FUNCTION FC_Concat4 : STRING
VAR_INPUT
    STR1: STRING(255);
    STR2: STRING(255);
    STR3: STRING(255):= '';
    STR4: STRING(255):= '';
    // etc up to a large number
END_VAR
VAR
	
END_VAR



FC_Concat4 := CONCAT(STR1 := FC_Concat4, STR2 := STR1);
FC_Concat4 := CONCAT(STR1 := FC_Concat4, STR2 := STR2);
FC_Concat4 := CONCAT(STR1 := FC_Concat4, STR2 := STR3);
FC_Concat4 := CONCAT(STR1 := FC_Concat4, STR2 := STR4);
// etc up to all defined inputs

END_FUNCTION

(* stored: Version 1.1.0.1, ProductVersion 3.1.4024.13
   POU FC_Concat4: Id {c0e2f29f-b3dc-4d20-9c67-5bbb16f4a64c}, SpecialFunc None *)
